Staubli VAL3: VelocityCmdMsg.dtx

public Header header
  [0]
    num nMsgType
    num nCommType
    num nReplyCode
    num nData[12]
public Body body
  [0]
    num nData[32]
public Prefix prefix
  [0]
    num nLength
    num nData[4]
public VelocityCmd velCmd
  [0]
    num nSeq
    num nVelVec[6]
    num nCmdType
